MOVL C09896 V=800.0 PL=0
MOVL C09897 V=800.0 PL=0
MOVL C09898 V=800.0 PL=0
MOVL C09899 V=800.0 PL=0
MOVL C09900 V=800.0 PL=0
MOVL C09901 V=800.0 PL=0
MOVL C09902 V=800.0 PL=0
MOVL C09903 V=800.0 PL=0
MOVL C09904 V=800.0 PL=0
MOVL C09905 V=800.0 PL=0
MOVL C09906 V=800.0 PL=0
MOVL C09907 V=800.0 PL=0
MOVL C09908 V=800.0 PL=0
MOVL C09909 V=800.0 PL=0
MOVL C09910 V=800.0 PL=0
MOVL C09911 V=800.0 PL=0
MOVL C09912 V=800.0 PL=0
MOVL C09913 V=800.0 PL=0
MOVL C09914 V=800.0 PL=0
MOVL C09915 V=800.0 PL=0
MOVL C09916 V=800.0 PL=0
MOVL C09917 V=800.0 PL=0
MOVL C09918 V=800.0 PL=0
MOVL C09919 V=800.0 PL=0
MOVL C09920 V=800.0 PL=0
MOVL C09921 V=800.0 PL=0
MOVL C09922 V=800.0 PL=0
MOVL C09923 V=800.0 PL=0
MOVL C09924 V=800.0 PL=0
MOVL C09925 V=800.0 PL=0
MOVL C09926 V=800.0 PL=0
MOVL C09927 V=800.0 PL=0
MOVL C09928 V=800.0 PL=0
MOVL C09929 V=800.0 PL=0
MOVL C09930 V=800.0 PL=0
MOVL C09931 V=800.0 PL=0
MOVL C09932 V=800.0 PL=0
MOVL C09933 V=800.0 PL=0
MOVL C09934 V=800.0 PL=0
MOVL C09935 V=800.0 PL=0
MOVL C09936 V=800.0 PL=0
MOVL C09937 V=800.0 PL=0
MOVL C09938 V=800.0 PL=0
MOVL C09939 V=800.0 PL=0
MOVL C09940 V=800.0 PL=0
MOVL C09941 V=800.0 PL=0
MOVL C09942 V=800.0 PL=0
MOVL C09943 V=800.0 PL=0
MOVL C09944 V=800.0 PL=0
MOVL C09945 V=800.0 PL=0
MOVL C09946 V=800.0 PL=0
MOVL C09947 V=800.0 PL=0
MOVL C09948 V=800.0 PL=0
MOVL C09949 V=800.0 PL=0
MOVL C09950 V=800.0 PL=0
MOVL C09951 V=800.0 PL=0
MOVL C09952 V=800.0 PL=0
MOVL C09953 V=800.0 PL=0
MOVL C09954 V=800.0 PL=0
MOVL C09955 V=800.0 PL=0
MOVL C09956 V=800.0 PL=0
MOVL C09957 V=800.0 PL=0
MOVL C09958 V=800.0 PL=0
MOVL C09959 V=800.0 PL=0
MOVL C09960 V=800.0 PL=0
MOVL C09961 V=800.0 PL=0
MOVL C09962 V=800.0 PL=0
MOVL C09963 V=800.0 PL=0
MOVL C09964 V=800.0 PL=0
MOVL C09965 V=800.0 PL=0
MOVL C09966 V=800.0 PL=0
MOVL C09967 V=800.0 PL=0
MOVL C09968 V=800.0 PL=0
MOVL C09969 V=800.0 PL=0
MOVL C09970 V=800.0 PL=0
MOVL C09971 V=800.0 PL=0
MOVL C09972 V=800.0 PL=0
MOVL C09973 V=800.0 PL=0
MOVL C09974 V=800.0 PL=0
MOVL C09975 V=800.0 PL=0
MOVL C09976 V=800.0 PL=0
MOVL C09977 V=800.0 PL=0
MOVL C09978 V=800.0 PL=0
MOVL C09979 V=800.0 PL=0
MOVL C09980 V=800.0 PL=0
MOVL C09981 V=800.0 PL=0
MOVL C09982 V=800.0 PL=0
MOVL C09983 V=800.0 PL=0
MOVL C09984 V=800.0 PL=0
MOVL C09985 V=800.0 PL=0
MOVL C09986 V=800.0 PL=0
MOVL C09987 V=800.0 PL=0
MOVL C09988 V=800.0 PL=0
MOVL C09989 V=800.0 PL=0
MOVL C09990 V=800.0 PL=0
MOVL C09991 V=800.0 PL=0
MOVL C09992 V=800.0 PL=0
MOVL C09993 V=800.0 PL=0
MOVL C09994 V=800.0 PL=0
MOVL C09995 V=800.0 PL=0
MOVL C09996 V=800.0 PL=0
CALL JOB:A_ROOF_SIDE_0617_2_PAINT_38
END
